FUNCTION_BLOCK FB_HeidConv
VAR_INPUT
	sHeidIn 			: STRING;
END_VAR
VAR_OUTPUT
	s1 					: STRING;
	s2 					: STRING;
	s3 					: STRING;
	s4 					: STRING;
END_VAR
VAR
	PosA 				: INT;
	PosB 				: INT;
	PosC 				: INT;
	PosD 				: INT;
	PosE 				: INT;
END_VAR

// Strip out "A" measurement"
PosA := FIND(sHeidIn, 'A');
PosB := FIND(sHeidIn, 'B');
s1 := sHeidIn;
s1 := DELETE(sHeidIn, LEN(sHeidIn) - PosB + 1, posB);
s1 := DELETE(s1, PosA, 1);


// Strip out "B" measurement
PosB := FIND(sHeidIn, 'B');
PosC := FIND(sHeidIn, 'C');
s2 := sHeidIn;
s2 := DELETE(sHeidIn, LEN(sHeidIn) - PosC + 1, PosC);
s2 := DELETE(s2, PosB, 1);

// Strip out "C" measurement"
PosC := FIND(sHeidIn, 'C');
PosD := FIND(sHeidIn, 'D');
s3 := sHeidIn;
s3 := DELETE(sHeidIn, LEN(sHeidIn) - PosD + 1, PosD);
s3 := DELETE(s3, PosC, 1);

// Strip out "D" measurement"
PosD := FIND(sHeidIn, 'D');
PosE := FIND(sHeidIn, 'E');
s4 := sHeidIn;
s4 := DELETE(sHeidIn, LEN(sHeidIn) - PosE + 1, PosE);
s4 := DELETE(s4, PosD, 1);

END_FUNCTION_BLOCK

(* stored: Version 1.1.0.1, ProductVersion 3.1.4024.2
   POU FB_HeidConv: Id {aaba04ae-91ec-4ea6-b44c-32fc3fd03f29}, SpecialFunc None *)
